FUNCTION_BLOCK ExampleDomain IMPLEMENTS I_DomainProvider, I_Execute
VAR_INPUT
END_VAR
VAR_OUTPUT
END_VAR
VAR CONSTANT
	MAX_STATE		: UDINT := 1;
END_VAR
VAR
	exe				: Execute(THIS^);

	// Context
	ctx				: ExampleDomain_Ctx;

	// State Machine
	
	stateMachine	: StateMachine;
	stateRepo		: StateRepo<MAX_STATE>;
	stateBuffer		: StateBuffer<MAX_STATE>;
	stateMgr		: StateManager<MAX_STATE>(stateMachine, stateRepo, stateBuffer);
	A_Smgr			: A_StateManager(stateMgr, ctx.priv.smgr);
	
	// States
	
	example			: ExampleDomain_ExampleState(stateRepo, ctx);
	exampleAssign	: A_Tag(example.Tag, ctx.state.iExample);
	
	// FLAGS
	flagList		: FlagList<0>;
	
	// SIGNALS
	signalList		: SignalList<0>;
	
	// RECEIVERS
	receiverList	: ReceiverList<0>;
	
	// HMI
	statusText		: ExampleDomain_StatusText(ctx);
	
	// DOMAIN
	domTag			: Tag;
	domain			: Domain(domTag, stateMgr, flagList, signalList, receiverList);
END_VAR

PROPERTY Dom : I_Domain
GET
Dom := domain;
END_GET
END_PROPERTY

METHOD Execute
END_METHOD

METHOD ToDebug : Debug.I_Debug
ToDebug := THIS^;
END_METHOD

END_FUNCTION_BLOCK

(* stored: Version 1.1.0.1
   POU ExampleDomain: Id {2cc7bbb1-01ad-4ca5-8dec-c2ca30454bb0}, SpecialFunc None
   Property Dom: Id {622704c3-9cc2-4725-8570-455b354fa60e}
   Get Get: Id {b38c86ed-180e-4b43-9a59-2077dac7971b}
   Method Execute: Id {c897e5cf-559a-456a-a239-6e33a3deb831}
   Method ToDebug: Id {16ff1ce0-9d29-4c22-be24-eb3a4d0ca553} *)
